// Mitsubishi GX Works2 project: WraptasticRobot   PLC: L02

// global labels: Global1
VAR_GLOBAL
  BrakeOutput AT Y2 : BOOL;
  Start AT X1043 : BOOL;
  ProgramOn AT Y3 : BOOL;
  Homing AT X1044 : BOOL;
  Home AT Y4 : BOOL;
  TestIn AT Y1041 : BOOL;
  TestInput AT X6 : BOOL;
  CallMasterJob AT Y1002 : BOOL;
  ExternalServoOn AT Y1001 : BOOL;
  ExternalStart AT Y1000 : BOOL;
  CallMaster AT X7 : BOOL;
  RobotOn AT X2 : BOOL;
  StartRobot AT X3 : BOOL;
  RobotReady AT Y0 : BOOL;
END_VAR

PROGRAM Robot
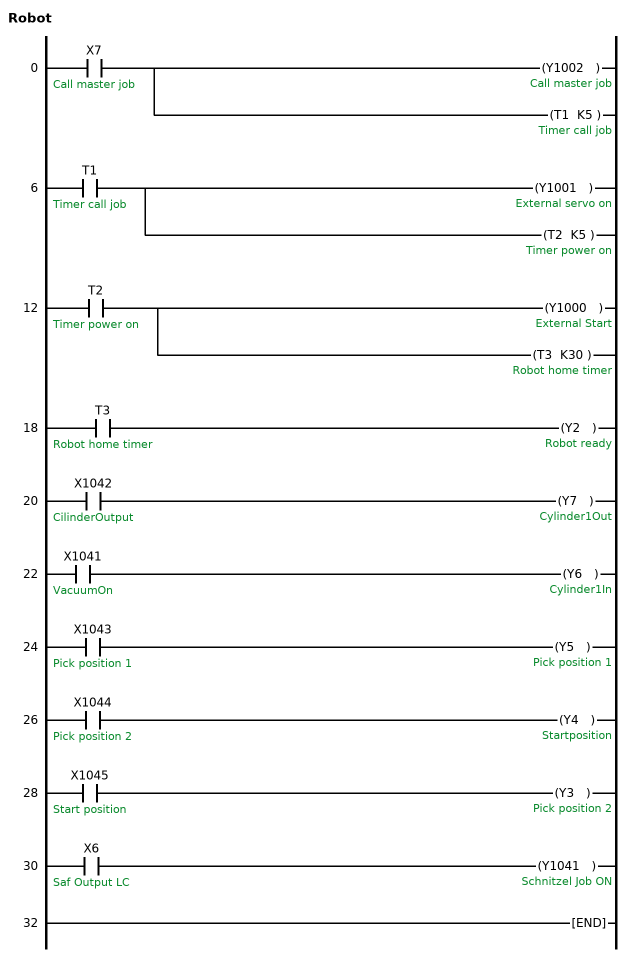
0     LD      X7  ; Call master job
      OUT     Y1002  ; Call master job
      OUT     T1 K5  ; Timer call job
6     LD      T1  ; Timer call job
      OUT     Y1001  ; External servo on
      OUT     T2 K5  ; Timer power on
12    LD      T2  ; Timer power on
      OUT     Y1000  ; External Start
      OUT     T3 K30  ; Robot home timer
18    LD      T3  ; Robot home timer
      OUT     Y2  ; Robot ready
20    LD      X1042  ; CilinderOutput
      OUT     Y7  ; Cylinder1Out
22    LD      X1041  ; VacuumOn
      OUT     Y6  ; Cylinder1In
24    LD      X1043  ; Pick position 1
      OUT     Y5  ; Pick position 1
26    LD      X1044  ; Pick position 2
      OUT     Y4  ; Startposition
28    LD      X1045  ; Start position
      OUT     Y3  ; Pick position 2
30    LD      X6  ; Saf Output LC
      OUT     Y1041  ; Schnitzel Job ON
32    END
END_PROGRAM

// device comments not shown above
Y0  ; RobotHome
